PROGRAM MAIN
VAR
END_VAR

//********************
// Command Pattern 
//********************
PRG_SampleCommandPattern();

END_PROGRAM

(* stored: Version 1.1.0.1
   POU MAIN: Id {e36a512e-fa25-440c-ad65-a91fa6a1270d}, SpecialFunc None *)
